PROGRAM PRG_Main
VAR
	fbMachine : FB_IndexedSiliconeMachine;
	tonHMIAliveOn        : TON;
    tonHMIAliveOff       : TON;
    bOutHMI   			 : BOOL;
	stCycleDataCSV     : ST_CycleDataCSV;
	bCycleDataCSVWrite : BOOL;
	
END_VAR

// Recommended task order:
// 1. PRG_IoMapping reads physical inputs at the beginning of the task.
// 2. PRG_HmiInterface builds application commands.
// 3. PRG_Main executes the reusable machine object.
// 4. PRG_HmiInterface publishes status.
// 5. PRG_IoMapping writes physical outputs at the end of the task.
ACT_UserLogout();

fbMachine.Cyclic(
    stInputs      := GVL_MASTER.stInputs,
    stCommand     := GVL_MASTER.stCommand,
    stConfig      := GVL_Config.stMachine,
    stIvekInput   := GVL_MASTER.stIvekInput,
    bIvekCommsOk  := GVL_MASTER.bIvekCommsOk,
	blogoutHMI 	  := bOutHMI,
    stOutputs     => GVL_MASTER.stOutputs,
    stStatus      => GVL_MASTER.stStatus,	
    stIvekOutput  => GVL_MASTER.stIvekOutput,
	stCycleDataCSVOut     => stCycleDataCSV,
	bCycleDataCSVWriteOut => bCycleDataCSVWrite);
	
	
D_1_PRG_CycleDataCSV.stCycleData := stCycleDataCSV;
D_1_PRG_CycleDataCSV.bWriteRequest := bCycleDataCSVWrite;

ACTION ACT_UserLogout:
tonHMIAliveOn(
    IN := GVL_HMI.bHMIAlive,
    PT := T#2S
);

tonHMIAliveOff(
    IN := NOT GVL_HMI.bHMIAlive,
    PT := T#2S
);

bOutHMI :=
    tonHMIAliveOn.Q
    OR tonHMIAliveOff.Q;
END_ACTION

END_PROGRAM

(* stored: Version 1.1.0.1, ProductVersion 3.1.4026.18
   POU PRG_Main: Id {f4d87ecd-c7bb-4ae4-b2e0-8161ff139d95}, SpecialFunc None
   Action ACT_UserLogout: Id {5c1cdba2-cfdc-4365-84bf-77af4bab5a6c} *)
